  PROC Part13()
    MoveL Offs(pOrigin,150.7,114.4,0.0),vDraw,z1,tPen\WObj:=wPaper;
    MoveL Offs(pOrigin,150.5,114.2,0.0),vDraw,z1,tPen\WObj:=wPaper;
    MoveL Offs(pOrigin,150.5,113.3,0.0),vDraw,z1,tPen\WObj:=wPaper;
    MoveL Offs(pOrigin,150.2,113.0,0.0),vDraw,z1,tPen\WObj:=wPaper;
    MoveL Offs(pOrigin,150.0,113.0,0.0),vDraw,z1,tPen\WObj:=wPaper;
    MoveL Offs(pOrigin,149.8,113.3,0.0),vDraw,z1,tPen\WObj:=wPaper;
    MoveL Offs(pOrigin,149.8,113.7,0.0),vDraw,z1,tPen\WObj:=wPaper;
    MoveL Offs(pOrigin,150.0,114.0,0.0),vDraw,z1,tPen\WObj:=wPaper;
    MoveL Offs(pOrigin,150.0,114.2,0.0),vDraw,z1,tPen\WObj:=wPaper;
    MoveL Offs(pOrigin,149.1,114.2,0.0),vDraw,z1,tPen\WObj:=wPaper;
    MoveL Offs(pOrigin,148.8,114.4,0.0),vDraw,z1,tPen\WObj:=wPaper;
    MoveL Offs(pOrigin,148.1,114.4,0.0),vDraw,z1,tPen\WObj:=wPaper;
    MoveL Offs(pOrigin,147.9,114.7,0.0),vDraw,z1,tPen\WObj:=wPaper;
    MoveL Offs(pOrigin,147.7,114.7,0.0),vDraw,z1,tPen\WObj:=wPaper;
    MoveL Offs(pOrigin,147.4,114.4,0.0),vDraw,z1,tPen\WObj:=wPaper;
    MoveL Offs(pOrigin,147.0,114.4,0.0),vDraw,z1,tPen\WObj:=wPaper;
    MoveL Offs(pOrigin,146.5,114.0,0.0),vDraw,z1,tPen\WObj:=wPaper;
    MoveL Offs(pOrigin,145.8,114.0,0.0),vDraw,z1,tPen\WObj:=wPaper;
    MoveL Offs(pOrigin,145.6,114.2,0.0),vDraw,z1,tPen\WObj:=wPaper;
    MoveL Offs(pOrigin,145.3,114.9,0.0),vDraw,z1,tPen\WObj:=wPaper;
    MoveL Offs(pOrigin,145.1,114.9,0.0),vDraw,z1,tPen\WObj:=wPaper;
    MoveL Offs(pOrigin,144.4,115.4,0.0),vDraw,z1,tPen\WObj:=wPaper;
    MoveL Offs(pOrigin,144.4,115.6,0.0),vDraw,z1,tPen\WObj:=wPaper;
    MoveL Offs(pOrigin,144.2,115.8,0.0),vDraw,z1,tPen\WObj:=wPaper;
    MoveL Offs(pOrigin,144.2,116.5,0.0),vDraw,z1,tPen\WObj:=wPaper;
    MoveL Offs(pOrigin,143.7,117.2,0.0),vDraw,z1,tPen\WObj:=wPaper;
    MoveL Offs(pOrigin,143.7,117.7,0.0),vDraw,z1,tPen\WObj:=wPaper;
    MoveL Offs(pOrigin,143.5,117.9,0.0),vDraw,z1,tPen\WObj:=wPaper;
    MoveL Offs(pOrigin,143.5,118.4,0.0),vDraw,z1,tPen\WObj:=wPaper;
    MoveL Offs(pOrigin,143.2,118.6,0.0),vDraw,z1,tPen\WObj:=wPaper;
    MoveL Offs(pOrigin,143.2,119.6,0.0),vDraw,z1,tPen\WObj:=wPaper;
    MoveL Offs(pOrigin,143.9,120.7,0.0),vDraw,z1,tPen\WObj:=wPaper;
    MoveL Offs(pOrigin,143.9,121.4,0.0),vDraw,z1,tPen\WObj:=wPaper;
    MoveL Offs(pOrigin,144.9,122.1,0.0),vDraw,z1,tPen\WObj:=wPaper;
    MoveL Offs(pOrigin,146.7,120.5,0.0),vDraw,z1,tPen\WObj:=wPaper;
    MoveL Offs(pOrigin,147.9,120.0,0.0),vDraw,z1,tPen\WObj:=wPaper;
    MoveL Offs(pOrigin,148.4,119.6,0.0),vDraw,z1,tPen\WObj:=wPaper;
    MoveL Offs(pOrigin,148.4,119.3,0.0),vDraw,z1,tPen\WObj:=wPaper;
    MoveL Offs(pOrigin,149.3,118.6,0.0),vDraw,fine,tPen\WObj:=wPaper;
    MoveL Offs(pOrigin,149.3,118.6,15.0),vApproach,z5,tPen\WObj:=wPaper;
    MoveL Offs(pOrigin,155.6,113.5,15.0),vTravel,z5,tPen\WObj:=wPaper;
    MoveL Offs(pOrigin,155.6,113.5,0.0),vApproach,fine,tPen\WObj:=wPaper;
    MoveL Offs(pOrigin,156.3,114.2,0.0),vDraw,z1,tPen\WObj:=wPaper;
    MoveL Offs(pOrigin,156.5,114.2,0.0),vDraw,z1,tPen\WObj:=wPaper;
    MoveL Offs(pOrigin,156.8,114.0,0.0),vDraw,z1,tPen\WObj:=wPaper;
    MoveL Offs(pOrigin,156.8,113.5,0.0),vDraw,z1,tPen\WObj:=wPaper;
    MoveL Offs(pOrigin,156.3,112.8,0.0),vDraw,z1,tPen\WObj:=wPaper;
    MoveL Offs(pOrigin,155.8,112.8,0.0),vDraw,z1,tPen\WObj:=wPaper;
    MoveL Offs(pOrigin,155.6,113.0,0.0),vDraw,z1,tPen\WObj:=wPaper;
    MoveL Offs(pOrigin,155.6,113.5,0.0),vDraw,fine,tPen\WObj:=wPaper;
    MoveL Offs(pOrigin,155.6,113.5,15.0),vApproach,z5,tPen\WObj:=wPaper;
    MoveL Offs(pOrigin,163.8,115.6,15.0),vTravel,z5,tPen\WObj:=wPaper;
    MoveL Offs(pOrigin,163.8,115.6,0.0),vApproach,fine,tPen\WObj:=wPaper;
    MoveL Offs(pOrigin,164.0,115.8,0.0),vDraw,z1,tPen\WObj:=wPaper;
    MoveL Offs(pOrigin,164.0,116.1,0.0),vDraw,z1,tPen\WObj:=wPaper;
    MoveL Offs(pOrigin,164.7,116.5,0.0),vDraw,z1,tPen\WObj:=wPaper;
    MoveL Offs(pOrigin,164.7,117.0,0.0),vDraw,z1,tPen\WObj:=wPaper;
    MoveL Offs(pOrigin,164.9,117.2,0.0),vDraw,z1,tPen\WObj:=wPaper;
    MoveL Offs(pOrigin,166.1,117.0,0.0),vDraw,z1,tPen\WObj:=wPaper;
    MoveL Offs(pOrigin,166.6,116.5,0.0),vDraw,z1,tPen\WObj:=wPaper;
    MoveL Offs(pOrigin,166.3,116.3,0.0),vDraw,z1,tPen\WObj:=wPaper;
    MoveL Offs(pOrigin,165.9,116.3,0.0),vDraw,z1,tPen\WObj:=wPaper;
    MoveL Offs(pOrigin,165.9,116.1,0.0),vDraw,z1,tPen\WObj:=wPaper;
    MoveL Offs(pOrigin,165.2,115.4,0.0),vDraw,z1,tPen\WObj:=wPaper;
    MoveL Offs(pOrigin,164.9,115.4,0.0),vDraw,z1,tPen\WObj:=wPaper;
    MoveL Offs(pOrigin,164.7,115.1,0.0),vDraw,z1,tPen\WObj:=wPaper;
    MoveL Offs(pOrigin,164.2,115.1,0.0),vDraw,z1,tPen\WObj:=wPaper;
    MoveL Offs(pOrigin,163.8,115.6,0.0),vDraw,fine,tPen\WObj:=wPaper;
    MoveL Offs(pOrigin,163.8,115.6,15.0),vApproach,z5,tPen\WObj:=wPaper;
    MoveL Offs(pOrigin,180.6,104.4,15.0),vTravel,z5,tPen\WObj:=wPaper;
    MoveL Offs(pOrigin,180.6,104.4,0.0),vApproach,fine,tPen\WObj:=wPaper;
    MoveL Offs(pOrigin,180.6,103.9,0.0),vDraw,z1,tPen\WObj:=wPaper;
    MoveL Offs(pOrigin,180.8,103.7,0.0),vDraw,z1,tPen\WObj:=wPaper;
    MoveL Offs(pOrigin,180.8,102.8,0.0),vDraw,z1,tPen\WObj:=wPaper;
    MoveL Offs(pOrigin,181.0,102.5,0.0),vDraw,z1,tPen\WObj:=wPaper;
    MoveL Offs(pOrigin,181.0,101.6,0.0),vDraw,z1,tPen\WObj:=wPaper;
    MoveL Offs(pOrigin,181.3,101.4,0.0),vDraw,z1,tPen\WObj:=wPaper;
    MoveL Offs(pOrigin,181.3,100.2,0.0),vDraw,z1,tPen\WObj:=wPaper;
    MoveL Offs(pOrigin,181.5,100.0,0.0),vDraw,z1,tPen\WObj:=wPaper;
    MoveL Offs(pOrigin,181.5,97.6,0.0),vDraw,z1,tPen\WObj:=wPaper;
    MoveL Offs(pOrigin,181.7,97.4,0.0),vDraw,z1,tPen\WObj:=wPaper;
    MoveL Offs(pOrigin,181.7,96.7,0.0),vDraw,z1,tPen\WObj:=wPaper;
    MoveL Offs(pOrigin,181.5,96.5,0.0),vDraw,z1,tPen\WObj:=wPaper;
    MoveL Offs(pOrigin,181.5,92.3,0.0),vDraw,z1,tPen\WObj:=wPaper;
    MoveL Offs(pOrigin,181.3,92.0,0.0),vDraw,z1,tPen\WObj:=wPaper;
    MoveL Offs(pOrigin,181.3,90.6,0.0),vDraw,z1,tPen\WObj:=wPaper;
    MoveL Offs(pOrigin,181.0,90.4,0.0),vDraw,z1,tPen\WObj:=wPaper;
    MoveL Offs(pOrigin,181.0,89.7,0.0),vDraw,z1,tPen\WObj:=wPaper;
    MoveL Offs(pOrigin,180.8,89.5,0.0),vDraw,z1,tPen\WObj:=wPaper;
    MoveL Offs(pOrigin,180.8,89.0,0.0),vDraw,z1,tPen\WObj:=wPaper;
    MoveL Offs(pOrigin,180.6,88.8,0.0),vDraw,z1,tPen\WObj:=wPaper;
    MoveL Offs(pOrigin,180.6,88.1,0.0),vDraw,z1,tPen\WObj:=wPaper;
    MoveL Offs(pOrigin,180.3,87.8,0.0),vDraw,z1,tPen\WObj:=wPaper;
    MoveL Offs(pOrigin,180.3,86.9,0.0),vDraw,z1,tPen\WObj:=wPaper;
    MoveL Offs(pOrigin,180.1,86.7,0.0),vDraw,z1,tPen\WObj:=wPaper;
    MoveL Offs(pOrigin,180.1,86.0,0.0),vDraw,z1,tPen\WObj:=wPaper;
    MoveL Offs(pOrigin,179.9,85.7,0.0),vDraw,z1,tPen\WObj:=wPaper;
    MoveL Offs(pOrigin,179.9,85.0,0.0),vDraw,z1,tPen\WObj:=wPaper;
    MoveL Offs(pOrigin,179.6,84.8,0.0),vDraw,z1,tPen\WObj:=wPaper;
    MoveL Offs(pOrigin,179.6,83.9,0.0),vDraw,z1,tPen\WObj:=wPaper;
    MoveL Offs(pOrigin,179.4,83.6,0.0),vDraw,z1,tPen\WObj:=wPaper;
    MoveL Offs(pOrigin,179.4,82.5,0.0),vDraw,z1,tPen\WObj:=wPaper;
    MoveL Offs(pOrigin,179.2,82.2,0.0),vDraw,z1,tPen\WObj:=wPaper;
    MoveL Offs(pOrigin,179.2,81.1,0.0),vDraw,z1,tPen\WObj:=wPaper;
    MoveL Offs(pOrigin,178.9,80.8,0.0),vDraw,z1,tPen\WObj:=wPaper;
    MoveL Offs(pOrigin,178.9,79.7,0.0),vDraw,z1,tPen\WObj:=wPaper;
    MoveL Offs(pOrigin,178.7,79.4,0.0),vDraw,z1,tPen\WObj:=wPaper;
    MoveL Offs(pOrigin,178.7,78.0,0.0),vDraw,z1,tPen\WObj:=wPaper;
    MoveL Offs(pOrigin,178.5,77.8,0.0),vDraw,z1,tPen\WObj:=wPaper;
    MoveL Offs(pOrigin,178.5,76.4,0.0),vDraw,z1,tPen\WObj:=wPaper;
    MoveL Offs(pOrigin,178.2,76.2,0.0),vDraw,z1,tPen\WObj:=wPaper;
    MoveL Offs(pOrigin,178.2,75.5,0.0),vDraw,z1,tPen\WObj:=wPaper;
    MoveL Offs(pOrigin,178.0,75.2,0.0),vDraw,z1,tPen\WObj:=wPaper;
    MoveL Offs(pOrigin,178.0,74.3,0.0),vDraw,z1,tPen\WObj:=wPaper;
    MoveL Offs(pOrigin,177.8,74.1,0.0),vDraw,z1,tPen\WObj:=wPaper;
    MoveL Offs(pOrigin,177.8,72.4,0.0),vDraw,z1,tPen\WObj:=wPaper;
    MoveL Offs(pOrigin,177.5,72.2,0.0),vDraw,z1,tPen\WObj:=wPaper;
    MoveL Offs(pOrigin,177.5,71.7,0.0),vDraw,z1,tPen\WObj:=wPaper;
    MoveL Offs(pOrigin,177.3,71.5,0.0),vDraw,z1,tPen\WObj:=wPaper;
    MoveL Offs(pOrigin,177.3,70.3,0.0),vDraw,z1,tPen\WObj:=wPaper;
  ENDPROC

  PROC Part14()
    MoveL Offs(pOrigin,177.1,70.1,0.0),vDraw,z1,tPen\WObj:=wPaper;
    MoveL Offs(pOrigin,177.1,69.2,0.0),vDraw,z1,tPen\WObj:=wPaper;
    MoveL Offs(pOrigin,176.8,68.9,0.0),vDraw,z1,tPen\WObj:=wPaper;
    MoveL Offs(pOrigin,176.8,67.8,0.0),vDraw,z1,tPen\WObj:=wPaper;
    MoveL Offs(pOrigin,176.6,67.5,0.0),vDraw,z1,tPen\WObj:=wPaper;
    MoveL Offs(pOrigin,176.6,66.4,0.0),vDraw,z1,tPen\WObj:=wPaper;
    MoveL Offs(pOrigin,176.4,66.1,0.0),vDraw,z1,tPen\WObj:=wPaper;
    MoveL Offs(pOrigin,176.4,65.2,0.0),vDraw,z1,tPen\WObj:=wPaper;
    MoveL Offs(pOrigin,176.1,65.0,0.0),vDraw,z1,tPen\WObj:=wPaper;
    MoveL Offs(pOrigin,176.1,64.0,0.0),vDraw,z1,tPen\WObj:=wPaper;
    MoveL Offs(pOrigin,175.9,63.8,0.0),vDraw,z1,tPen\WObj:=wPaper;
    MoveL Offs(pOrigin,175.9,62.6,0.0),vDraw,z1,tPen\WObj:=wPaper;
    MoveL Offs(pOrigin,175.7,62.4,0.0),vDraw,z1,tPen\WObj:=wPaper;
    MoveL Offs(pOrigin,175.7,61.5,0.0),vDraw,z1,tPen\WObj:=wPaper;
    MoveL Offs(pOrigin,175.4,61.2,0.0),vDraw,z1,tPen\WObj:=wPaper;
    MoveL Offs(pOrigin,175.4,60.5,0.0),vDraw,z1,tPen\WObj:=wPaper;
    MoveL Offs(pOrigin,175.2,60.3,0.0),vDraw,z1,tPen\WObj:=wPaper;
    MoveL Offs(pOrigin,175.2,59.1,0.0),vDraw,z1,tPen\WObj:=wPaper;
    MoveL Offs(pOrigin,175.0,58.9,0.0),vDraw,z1,tPen\WObj:=wPaper;
    MoveL Offs(pOrigin,175.0,58.0,0.0),vDraw,z1,tPen\WObj:=wPaper;
    MoveL Offs(pOrigin,174.7,57.7,0.0),vDraw,z1,tPen\WObj:=wPaper;
    MoveL Offs(pOrigin,174.7,57.0,0.0),vDraw,z1,tPen\WObj:=wPaper;
    MoveL Offs(pOrigin,174.5,56.8,0.0),vDraw,z1,tPen\WObj:=wPaper;
    MoveL Offs(pOrigin,174.5,55.9,0.0),vDraw,z1,tPen\WObj:=wPaper;
    MoveL Offs(pOrigin,174.3,55.6,0.0),vDraw,z1,tPen\WObj:=wPaper;
    MoveL Offs(pOrigin,174.3,54.7,0.0),vDraw,z1,tPen\WObj:=wPaper;
    MoveL Offs(pOrigin,174.0,54.5,0.0),vDraw,z1,tPen\WObj:=wPaper;
    MoveL Offs(pOrigin,174.0,53.8,0.0),vDraw,z1,tPen\WObj:=wPaper;
    MoveL Offs(pOrigin,173.8,53.5,0.0),vDraw,z1,tPen\WObj:=wPaper;
    MoveL Offs(pOrigin,173.8,52.6,0.0),vDraw,z1,tPen\WObj:=wPaper;
    MoveL Offs(pOrigin,173.6,52.4,0.0),vDraw,z1,tPen\WObj:=wPaper;
    MoveL Offs(pOrigin,173.6,51.7,0.0),vDraw,z1,tPen\WObj:=wPaper;
    MoveL Offs(pOrigin,173.3,51.4,0.0),vDraw,z1,tPen\WObj:=wPaper;
    MoveL Offs(pOrigin,173.3,50.5,0.0),vDraw,z1,tPen\WObj:=wPaper;
    MoveL Offs(pOrigin,173.1,50.3,0.0),vDraw,z1,tPen\WObj:=wPaper;
    MoveL Offs(pOrigin,173.1,49.6,0.0),vDraw,z1,tPen\WObj:=wPaper;
    MoveL Offs(pOrigin,172.9,49.3,0.0),vDraw,z1,tPen\WObj:=wPaper;
    MoveL Offs(pOrigin,172.9,48.4,0.0),vDraw,z1,tPen\WObj:=wPaper;
    MoveL Offs(pOrigin,172.6,48.2,0.0),vDraw,z1,tPen\WObj:=wPaper;
    MoveL Offs(pOrigin,172.6,47.2,0.0),vDraw,z1,tPen\WObj:=wPaper;
    MoveL Offs(pOrigin,172.4,47.0,0.0),vDraw,z1,tPen\WObj:=wPaper;
    MoveL Offs(pOrigin,172.4,46.1,0.0),vDraw,z1,tPen\WObj:=wPaper;
    MoveL Offs(pOrigin,172.2,45.8,0.0),vDraw,z1,tPen\WObj:=wPaper;
    MoveL Offs(pOrigin,172.2,44.9,0.0),vDraw,z1,tPen\WObj:=wPaper;
    MoveL Offs(pOrigin,171.9,44.7,0.0),vDraw,z1,tPen\WObj:=wPaper;
    MoveL Offs(pOrigin,171.9,44.0,0.0),vDraw,z1,tPen\WObj:=wPaper;
    MoveL Offs(pOrigin,171.7,43.7,0.0),vDraw,z1,tPen\WObj:=wPaper;
    MoveL Offs(pOrigin,171.7,43.0,0.0),vDraw,z1,tPen\WObj:=wPaper;
    MoveL Offs(pOrigin,171.5,42.8,0.0),vDraw,z1,tPen\WObj:=wPaper;
    MoveL Offs(pOrigin,171.5,41.9,0.0),vDraw,z1,tPen\WObj:=wPaper;
    MoveL Offs(pOrigin,171.2,41.6,0.0),vDraw,z1,tPen\WObj:=wPaper;
    MoveL Offs(pOrigin,171.2,40.9,0.0),vDraw,z1,tPen\WObj:=wPaper;
    MoveL Offs(pOrigin,171.0,40.7,0.0),vDraw,z1,tPen\WObj:=wPaper;
    MoveL Offs(pOrigin,171.0,39.8,0.0),vDraw,z1,tPen\WObj:=wPaper;
    MoveL Offs(pOrigin,170.8,39.5,0.0),vDraw,z1,tPen\WObj:=wPaper;
    MoveL Offs(pOrigin,170.8,38.8,0.0),vDraw,z1,tPen\WObj:=wPaper;
    MoveL Offs(pOrigin,170.5,38.6,0.0),vDraw,z1,tPen\WObj:=wPaper;
    MoveL Offs(pOrigin,170.5,37.7,0.0),vDraw,z1,tPen\WObj:=wPaper;
    MoveL Offs(pOrigin,170.3,37.4,0.0),vDraw,z1,tPen\WObj:=wPaper;
    MoveL Offs(pOrigin,170.3,36.7,0.0),vDraw,z1,tPen\WObj:=wPaper;
    MoveL Offs(pOrigin,170.1,36.5,0.0),vDraw,z1,tPen\WObj:=wPaper;
    MoveL Offs(pOrigin,170.1,35.8,0.0),vDraw,z1,tPen\WObj:=wPaper;
    MoveL Offs(pOrigin,169.8,35.6,0.0),vDraw,z1,tPen\WObj:=wPaper;
    MoveL Offs(pOrigin,169.8,34.9,0.0),vDraw,z1,tPen\WObj:=wPaper;
    MoveL Offs(pOrigin,169.6,34.6,0.0),vDraw,z1,tPen\WObj:=wPaper;
    MoveL Offs(pOrigin,169.6,33.7,0.0),vDraw,z1,tPen\WObj:=wPaper;
    MoveL Offs(pOrigin,169.4,33.5,0.0),vDraw,z1,tPen\WObj:=wPaper;
    MoveL Offs(pOrigin,169.4,32.8,0.0),vDraw,z1,tPen\WObj:=wPaper;
    MoveL Offs(pOrigin,169.1,32.5,0.0),vDraw,z1,tPen\WObj:=wPaper;
    MoveL Offs(pOrigin,169.1,31.8,0.0),vDraw,z1,tPen\WObj:=wPaper;
    MoveL Offs(pOrigin,168.9,31.6,0.0),vDraw,z1,tPen\WObj:=wPaper;
    MoveL Offs(pOrigin,168.9,30.9,0.0),vDraw,z1,tPen\WObj:=wPaper;
    MoveL Offs(pOrigin,168.7,30.7,0.0),vDraw,z1,tPen\WObj:=wPaper;
    MoveL Offs(pOrigin,168.7,29.7,0.0),vDraw,z1,tPen\WObj:=wPaper;
    MoveL Offs(pOrigin,168.4,29.5,0.0),vDraw,z1,tPen\WObj:=wPaper;
    MoveL Offs(pOrigin,168.4,28.8,0.0),vDraw,z1,tPen\WObj:=wPaper;
    MoveL Offs(pOrigin,168.2,28.6,0.0),vDraw,z1,tPen\WObj:=wPaper;
    MoveL Offs(pOrigin,168.2,27.6,0.0),vDraw,z1,tPen\WObj:=wPaper;
    MoveL Offs(pOrigin,168.0,27.4,0.0),vDraw,z1,tPen\WObj:=wPaper;
    MoveL Offs(pOrigin,168.0,26.9,0.0),vDraw,z1,tPen\WObj:=wPaper;
    MoveL Offs(pOrigin,167.7,26.7,0.0),vDraw,z1,tPen\WObj:=wPaper;
    MoveL Offs(pOrigin,167.7,25.8,0.0),vDraw,z1,tPen\WObj:=wPaper;
    MoveL Offs(pOrigin,167.5,25.5,0.0),vDraw,z1,tPen\WObj:=wPaper;
    MoveL Offs(pOrigin,167.5,24.8,0.0),vDraw,z1,tPen\WObj:=wPaper;
    MoveL Offs(pOrigin,167.3,24.6,0.0),vDraw,z1,tPen\WObj:=wPaper;
    MoveL Offs(pOrigin,167.3,23.9,0.0),vDraw,z1,tPen\WObj:=wPaper;
    MoveL Offs(pOrigin,167.0,23.7,0.0),vDraw,z1,tPen\WObj:=wPaper;
    MoveL Offs(pOrigin,167.0,23.0,0.0),vDraw,z1,tPen\WObj:=wPaper;
    MoveL Offs(pOrigin,166.8,22.7,0.0),vDraw,z1,tPen\WObj:=wPaper;
    MoveL Offs(pOrigin,166.8,22.0,0.0),vDraw,z1,tPen\WObj:=wPaper;
    MoveL Offs(pOrigin,166.6,21.8,0.0),vDraw,z1,tPen\WObj:=wPaper;
    MoveL Offs(pOrigin,166.6,21.1,0.0),vDraw,z1,tPen\WObj:=wPaper;
    MoveL Offs(pOrigin,166.3,20.9,0.0),vDraw,z1,tPen\WObj:=wPaper;
    MoveL Offs(pOrigin,166.3,20.2,0.0),vDraw,z1,tPen\WObj:=wPaper;
    MoveL Offs(pOrigin,166.1,19.9,0.0),vDraw,z1,tPen\WObj:=wPaper;
    MoveL Offs(pOrigin,166.1,19.5,0.0),vDraw,z1,tPen\WObj:=wPaper;
    MoveL Offs(pOrigin,165.9,19.2,0.0),vDraw,z1,tPen\WObj:=wPaper;
    MoveL Offs(pOrigin,165.9,18.3,0.0),vDraw,z1,tPen\WObj:=wPaper;
    MoveL Offs(pOrigin,165.6,18.1,0.0),vDraw,z1,tPen\WObj:=wPaper;
    MoveL Offs(pOrigin,165.6,17.6,0.0),vDraw,z1,tPen\WObj:=wPaper;
    MoveL Offs(pOrigin,165.4,17.4,0.0),vDraw,z1,tPen\WObj:=wPaper;
    MoveL Offs(pOrigin,165.4,16.7,0.0),vDraw,z1,tPen\WObj:=wPaper;
    MoveL Offs(pOrigin,165.2,16.4,0.0),vDraw,z1,tPen\WObj:=wPaper;
    MoveL Offs(pOrigin,165.2,15.7,0.0),vDraw,z1,tPen\WObj:=wPaper;
    MoveL Offs(pOrigin,164.9,15.5,0.0),vDraw,z1,tPen\WObj:=wPaper;
    MoveL Offs(pOrigin,164.9,14.8,0.0),vDraw,z1,tPen\WObj:=wPaper;
    MoveL Offs(pOrigin,164.7,14.6,0.0),vDraw,z1,tPen\WObj:=wPaper;
    MoveL Offs(pOrigin,164.7,13.9,0.0),vDraw,z1,tPen\WObj:=wPaper;
    MoveL Offs(pOrigin,164.5,13.6,0.0),vDraw,z1,tPen\WObj:=wPaper;
    MoveL Offs(pOrigin,164.5,12.9,0.0),vDraw,z1,tPen\WObj:=wPaper;
    MoveL Offs(pOrigin,164.2,12.7,0.0),vDraw,z1,tPen\WObj:=wPaper;
    MoveL Offs(pOrigin,164.2,12.0,0.0),vDraw,z1,tPen\WObj:=wPaper;
    MoveL Offs(pOrigin,164.0,11.8,0.0),vDraw,z1,tPen\WObj:=wPaper;
    MoveL Offs(pOrigin,164.0,11.1,0.0),vDraw,z1,tPen\WObj:=wPaper;
    MoveL Offs(pOrigin,163.8,10.8,0.0),vDraw,z1,tPen\WObj:=wPaper;
    MoveL Offs(pOrigin,163.8,10.1,0.0),vDraw,z1,tPen\WObj:=wPaper;
    MoveL Offs(pOrigin,163.5,9.9,0.0),vDraw,z1,tPen\WObj:=wPaper;
    MoveL Offs(pOrigin,163.5,9.4,0.0),vDraw,z1,tPen\WObj:=wPaper;
    MoveL Offs(pOrigin,163.3,9.2,0.0),vDraw,z1,tPen\WObj:=wPaper;
    MoveL Offs(pOrigin,163.3,8.5,0.0),vDraw,z1,tPen\WObj:=wPaper;
  ENDPROC

  PROC Part15()
    MoveL Offs(pOrigin,163.1,8.3,0.0),vDraw,z1,tPen\WObj:=wPaper;
    MoveL Offs(pOrigin,163.1,7.6,0.0),vDraw,z1,tPen\WObj:=wPaper;
    MoveL Offs(pOrigin,162.8,7.3,0.0),vDraw,z1,tPen\WObj:=wPaper;
    MoveL Offs(pOrigin,162.8,6.6,0.0),vDraw,z1,tPen\WObj:=wPaper;
    MoveL Offs(pOrigin,162.6,6.4,0.0),vDraw,z1,tPen\WObj:=wPaper;
    MoveL Offs(pOrigin,162.6,5.7,0.0),vDraw,z1,tPen\WObj:=wPaper;
    MoveL Offs(pOrigin,162.4,5.5,0.0),vDraw,z1,tPen\WObj:=wPaper;
    MoveL Offs(pOrigin,162.4,5.2,0.0),vDraw,z1,tPen\WObj:=wPaper;
    MoveL Offs(pOrigin,231.7,5.2,0.0),vDraw,z1,tPen\WObj:=wPaper;
    MoveL Offs(pOrigin,231.7,78.5,0.0),vDraw,z1,tPen\WObj:=wPaper;
    MoveL Offs(pOrigin,230.7,78.5,0.0),vDraw,z1,tPen\WObj:=wPaper;
    MoveL Offs(pOrigin,230.5,78.3,0.0),vDraw,z1,tPen\WObj:=wPaper;
    MoveL Offs(pOrigin,230.0,78.3,0.0),vDraw,z1,tPen\WObj:=wPaper;
    MoveL Offs(pOrigin,229.3,79.0,0.0),vDraw,z1,tPen\WObj:=wPaper;
    MoveL Offs(pOrigin,229.1,79.0,0.0),vDraw,z1,tPen\WObj:=wPaper;
    MoveL Offs(pOrigin,227.0,80.1,0.0),vDraw,z1,tPen\WObj:=wPaper;
    MoveL Offs(pOrigin,226.5,80.1,0.0),vDraw,z1,tPen\WObj:=wPaper;
    MoveL Offs(pOrigin,225.4,80.8,0.0),vDraw,z1,tPen\WObj:=wPaper;
    MoveL Offs(pOrigin,224.9,80.8,0.0),vDraw,z1,tPen\WObj:=wPaper;
    MoveL Offs(pOrigin,224.2,81.3,0.0),vDraw,z1,tPen\WObj:=wPaper;
    MoveL Offs(pOrigin,223.7,81.3,0.0),vDraw,z1,tPen\WObj:=wPaper;
    MoveL Offs(pOrigin,223.0,81.8,0.0),vDraw,z1,tPen\WObj:=wPaper;
    MoveL Offs(pOrigin,222.6,81.8,0.0),vDraw,z1,tPen\WObj:=wPaper;
    MoveL Offs(pOrigin,222.3,82.0,0.0),vDraw,z1,tPen\WObj:=wPaper;
    MoveL Offs(pOrigin,222.1,82.0,0.0),vDraw,z1,tPen\WObj:=wPaper;
    MoveL Offs(pOrigin,221.4,82.5,0.0),vDraw,z1,tPen\WObj:=wPaper;
    MoveL Offs(pOrigin,220.9,82.5,0.0),vDraw,z1,tPen\WObj:=wPaper;
    MoveL Offs(pOrigin,220.2,82.9,0.0),vDraw,z1,tPen\WObj:=wPaper;
    MoveL Offs(pOrigin,219.1,83.2,0.0),vDraw,z1,tPen\WObj:=wPaper;
    MoveL Offs(pOrigin,218.4,83.6,0.0),vDraw,z1,tPen\WObj:=wPaper;
    MoveL Offs(pOrigin,217.2,83.9,0.0),vDraw,z1,tPen\WObj:=wPaper;
    MoveL Offs(pOrigin,216.5,84.3,0.0),vDraw,z1,tPen\WObj:=wPaper;
    MoveL Offs(pOrigin,216.0,84.3,0.0),vDraw,z1,tPen\WObj:=wPaper;
    MoveL Offs(pOrigin,215.3,84.8,0.0),vDraw,z1,tPen\WObj:=wPaper;
    MoveL Offs(pOrigin,214.9,84.8,0.0),vDraw,z1,tPen\WObj:=wPaper;
    MoveL Offs(pOrigin,214.6,85.0,0.0),vDraw,z1,tPen\WObj:=wPaper;
    MoveL Offs(pOrigin,213.5,85.3,0.0),vDraw,z1,tPen\WObj:=wPaper;
    MoveL Offs(pOrigin,212.8,85.7,0.0),vDraw,z1,tPen\WObj:=wPaper;
    MoveL Offs(pOrigin,212.3,85.7,0.0),vDraw,z1,tPen\WObj:=wPaper;
    MoveL Offs(pOrigin,212.1,86.0,0.0),vDraw,z1,tPen\WObj:=wPaper;
    MoveL Offs(pOrigin,210.9,86.2,0.0),vDraw,z1,tPen\WObj:=wPaper;
    MoveL Offs(pOrigin,210.2,86.7,0.0),vDraw,z1,tPen\WObj:=wPaper;
    MoveL Offs(pOrigin,209.7,86.7,0.0),vDraw,z1,tPen\WObj:=wPaper;
    MoveL Offs(pOrigin,209.5,86.9,0.0),vDraw,z1,tPen\WObj:=wPaper;
    MoveL Offs(pOrigin,208.3,87.1,0.0),vDraw,z1,tPen\WObj:=wPaper;
    MoveL Offs(pOrigin,207.6,87.6,0.0),vDraw,z1,tPen\WObj:=wPaper;
    MoveL Offs(pOrigin,207.2,87.6,0.0),vDraw,z1,tPen\WObj:=wPaper;
    MoveL Offs(pOrigin,206.9,87.8,0.0),vDraw,z1,tPen\WObj:=wPaper;
    MoveL Offs(pOrigin,205.8,88.1,0.0),vDraw,z1,tPen\WObj:=wPaper;
    MoveL Offs(pOrigin,205.5,88.3,0.0),vDraw,z1,tPen\WObj:=wPaper;
    MoveL Offs(pOrigin,205.3,88.3,0.0),vDraw,z1,tPen\WObj:=wPaper;
    MoveL Offs(pOrigin,205.1,88.5,0.0),vDraw,z1,tPen\WObj:=wPaper;
    MoveL Offs(pOrigin,204.6,88.5,0.0),vDraw,z1,tPen\WObj:=wPaper;
    MoveL Offs(pOrigin,203.9,89.0,0.0),vDraw,z1,tPen\WObj:=wPaper;
    MoveL Offs(pOrigin,203.4,89.0,0.0),vDraw,z1,tPen\WObj:=wPaper;
    MoveL Offs(pOrigin,203.2,89.2,0.0),vDraw,z1,tPen\WObj:=wPaper;
    MoveL Offs(pOrigin,202.7,89.2,0.0),vDraw,z1,tPen\WObj:=wPaper;
    MoveL Offs(pOrigin,202.0,89.7,0.0),vDraw,z1,tPen\WObj:=wPaper;
    MoveL Offs(pOrigin,200.9,89.9,0.0),vDraw,z1,tPen\WObj:=wPaper;
    MoveL Offs(pOrigin,200.2,90.4,0.0),vDraw,z1,tPen\WObj:=wPaper;
    MoveL Offs(pOrigin,199.7,90.4,0.0),vDraw,z1,tPen\WObj:=wPaper;
    MoveL Offs(pOrigin,199.0,90.9,0.0),vDraw,z1,tPen\WObj:=wPaper;
    MoveL Offs(pOrigin,198.5,90.9,0.0),vDraw,z1,tPen\WObj:=wPaper;
    MoveL Offs(pOrigin,198.3,91.1,0.0),vDraw,z1,tPen\WObj:=wPaper;
    MoveL Offs(pOrigin,197.8,91.1,0.0),vDraw,z1,tPen\WObj:=wPaper;
    MoveL Offs(pOrigin,197.1,91.6,0.0),vDraw,z1,tPen\WObj:=wPaper;
    MoveL Offs(pOrigin,196.0,91.8,0.0),vDraw,z1,tPen\WObj:=wPaper;
    MoveL Offs(pOrigin,195.3,92.3,0.0),vDraw,z1,tPen\WObj:=wPaper;
    MoveL Offs(pOrigin,194.1,92.5,0.0),vDraw,z1,tPen\WObj:=wPaper;
    MoveL Offs(pOrigin,193.4,93.0,0.0),vDraw,z1,tPen\WObj:=wPaper;
    MoveL Offs(pOrigin,192.9,93.0,0.0),vDraw,z1,tPen\WObj:=wPaper;
    MoveL Offs(pOrigin,192.7,93.2,0.0),vDraw,z1,tPen\WObj:=wPaper;
    MoveL Offs(pOrigin,191.5,93.4,0.0),vDraw,z1,tPen\WObj:=wPaper;
    MoveL Offs(pOrigin,191.1,93.9,0.0),vDraw,z1,tPen\WObj:=wPaper;
    MoveL Offs(pOrigin,190.8,93.9,0.0),vDraw,z1,tPen\WObj:=wPaper;
    MoveL Offs(pOrigin,189.9,94.8,0.0),vDraw,z1,tPen\WObj:=wPaper;
    MoveL Offs(pOrigin,189.7,94.8,0.0),vDraw,z1,tPen\WObj:=wPaper;
    MoveL Offs(pOrigin,189.0,95.5,0.0),vDraw,z1,tPen\WObj:=wPaper;
    MoveL Offs(pOrigin,188.7,95.5,0.0),vDraw,z1,tPen\WObj:=wPaper;
    MoveL Offs(pOrigin,187.3,96.9,0.0),vDraw,z1,tPen\WObj:=wPaper;
    MoveL Offs(pOrigin,187.1,96.9,0.0),vDraw,z1,tPen\WObj:=wPaper;
    MoveL Offs(pOrigin,184.1,100.0,0.0),vDraw,z1,tPen\WObj:=wPaper;
    MoveL Offs(pOrigin,184.1,100.2,0.0),vDraw,z1,tPen\WObj:=wPaper;
    MoveL Offs(pOrigin,182.9,101.6,0.0),vDraw,z1,tPen\WObj:=wPaper;
    MoveL Offs(pOrigin,182.7,102.3,0.0),vDraw,z1,tPen\WObj:=wPaper;
    MoveL Offs(pOrigin,182.0,103.0,0.0),vDraw,z1,tPen\WObj:=wPaper;
    MoveL Offs(pOrigin,182.0,103.2,0.0),vDraw,z1,tPen\WObj:=wPaper;
    MoveL Offs(pOrigin,181.3,103.9,0.0),vDraw,z1,tPen\WObj:=wPaper;
    MoveL Offs(pOrigin,181.3,104.2,0.0),vDraw,z1,tPen\WObj:=wPaper;
    MoveL Offs(pOrigin,181.0,104.4,0.0),vDraw,z1,tPen\WObj:=wPaper;
    MoveL Offs(pOrigin,180.6,104.4,0.0),vDraw,fine,tPen\WObj:=wPaper;
    MoveL Offs(pOrigin,180.6,104.4,15.0),vApproach,z5,tPen\WObj:=wPaper;
    MoveL Offs(pOrigin,154.9,77.3,15.0),vTravel,z5,tPen\WObj:=wPaper;
    MoveL Offs(pOrigin,154.9,77.3,0.0),vApproach,fine,tPen\WObj:=wPaper;
    MoveL Offs(pOrigin,155.4,76.9,0.0),vDraw,z1,tPen\WObj:=wPaper;
    MoveL Offs(pOrigin,155.4,76.4,0.0),vDraw,z1,tPen\WObj:=wPaper;
    MoveL Offs(pOrigin,155.1,76.2,0.0),vDraw,z1,tPen\WObj:=wPaper;
    MoveL Offs(pOrigin,154.7,76.2,0.0),vDraw,z1,tPen\WObj:=wPaper;
    MoveL Offs(pOrigin,154.4,76.4,0.0),vDraw,z1,tPen\WObj:=wPaper;
    MoveL Offs(pOrigin,154.4,77.1,0.0),vDraw,z1,tPen\WObj:=wPaper;
    MoveL Offs(pOrigin,154.7,77.3,0.0),vDraw,z1,tPen\WObj:=wPaper;
    MoveL Offs(pOrigin,154.9,77.3,0.0),vDraw,fine,tPen\WObj:=wPaper;
    MoveL Offs(pOrigin,154.9,77.3,15.0),vApproach,z5,tPen\WObj:=wPaper;
    MoveL Offs(pOrigin,153.0,76.4,15.0),vTravel,z5,tPen\WObj:=wPaper;
    MoveL Offs(pOrigin,153.0,76.4,0.0),vApproach,fine,tPen\WObj:=wPaper;
    MoveL Offs(pOrigin,153.0,76.2,0.0),vDraw,z1,tPen\WObj:=wPaper;
    MoveL Offs(pOrigin,152.8,75.9,0.0),vDraw,z1,tPen\WObj:=wPaper;
    MoveL Offs(pOrigin,152.1,76.2,0.0),vDraw,z1,tPen\WObj:=wPaper;
    MoveL Offs(pOrigin,151.4,76.9,0.0),vDraw,z1,tPen\WObj:=wPaper;
    MoveL Offs(pOrigin,151.4,77.1,0.0),vDraw,z1,tPen\WObj:=wPaper;
    MoveL Offs(pOrigin,151.9,77.6,0.0),vDraw,z1,tPen\WObj:=wPaper;
    MoveL Offs(pOrigin,152.1,77.6,0.0),vDraw,z1,tPen\WObj:=wPaper;
    MoveL Offs(pOrigin,152.6,77.1,0.0),vDraw,z1,tPen\WObj:=wPaper;
    MoveL Offs(pOrigin,152.6,76.9,0.0),vDraw,z1,tPen\WObj:=wPaper;
    MoveL Offs(pOrigin,153.0,76.4,0.0),vDraw,fine,tPen\WObj:=wPaper;
    MoveL Offs(pOrigin,153.0,76.4,15.0),vApproach,z5,tPen\WObj:=wPaper;
    MoveL Offs(pOrigin,148.4,82.9,15.0),vTravel,z5,tPen\WObj:=wPaper;
    MoveL Offs(pOrigin,148.4,82.9,0.0),vApproach,fine,tPen\WObj:=wPaper;
    MoveL Offs(pOrigin,147.4,82.9,0.0),vDraw,z1,tPen\WObj:=wPaper;
    MoveL Offs(pOrigin,147.0,83.4,0.0),vDraw,z1,tPen\WObj:=wPaper;
  ENDPROC

  PROC Part16()
    MoveL Offs(pOrigin,147.0,83.9,0.0),vDraw,z1,tPen\WObj:=wPaper;
    MoveL Offs(pOrigin,147.2,84.1,0.0),vDraw,z1,tPen\WObj:=wPaper;
    MoveL Offs(pOrigin,147.2,84.3,0.0),vDraw,z1,tPen\WObj:=wPaper;
    MoveL Offs(pOrigin,147.0,84.6,0.0),vDraw,z1,tPen\WObj:=wPaper;
    MoveL Offs(pOrigin,147.0,85.0,0.0),vDraw,z1,tPen\WObj:=wPaper;
    MoveL Offs(pOrigin,146.7,85.3,0.0),vDraw,z1,tPen\WObj:=wPaper;
    MoveL Offs(pOrigin,146.0,85.3,0.0),vDraw,z1,tPen\WObj:=wPaper;
    MoveL Offs(pOrigin,145.6,84.8,0.0),vDraw,z1,tPen\WObj:=wPaper;
    MoveL Offs(pOrigin,144.9,84.8,0.0),vDraw,z1,tPen\WObj:=wPaper;
    MoveL Offs(pOrigin,144.6,85.0,0.0),vDraw,z1,tPen\WObj:=wPaper;
    MoveL Offs(pOrigin,144.4,85.0,0.0),vDraw,z1,tPen\WObj:=wPaper;
    MoveL Offs(pOrigin,143.2,86.2,0.0),vDraw,z1,tPen\WObj:=wPaper;
    MoveL Offs(pOrigin,143.0,86.2,0.0),vDraw,z1,tPen\WObj:=wPaper;
    MoveL Offs(pOrigin,142.5,86.7,0.0),vDraw,z1,tPen\WObj:=wPaper;
    MoveL Offs(pOrigin,142.1,86.7,0.0),vDraw,z1,tPen\WObj:=wPaper;
    MoveL Offs(pOrigin,140.0,89.0,0.0),vDraw,z1,tPen\WObj:=wPaper;
    MoveL Offs(pOrigin,140.0,89.2,0.0),vDraw,z1,tPen\WObj:=wPaper;
    MoveL Offs(pOrigin,139.7,89.5,0.0),vDraw,z1,tPen\WObj:=wPaper;
    MoveL Offs(pOrigin,139.7,89.9,0.0),vDraw,z1,tPen\WObj:=wPaper;
    MoveL Offs(pOrigin,140.0,90.2,0.0),vDraw,z1,tPen\WObj:=wPaper;
    MoveL Offs(pOrigin,140.2,90.2,0.0),vDraw,z1,tPen\WObj:=wPaper;
    MoveL Offs(pOrigin,140.4,89.9,0.0),vDraw,z1,tPen\WObj:=wPaper;
    MoveL Offs(pOrigin,141.1,89.9,0.0),vDraw,z1,tPen\WObj:=wPaper;
    MoveL Offs(pOrigin,141.6,89.5,0.0),vDraw,z1,tPen\WObj:=wPaper;
    MoveL Offs(pOrigin,142.3,89.2,0.0),vDraw,z1,tPen\WObj:=wPaper;
    MoveL Offs(pOrigin,143.5,88.1,0.0),vDraw,z1,tPen\WObj:=wPaper;
    MoveL Offs(pOrigin,144.2,87.8,0.0),vDraw,z1,tPen\WObj:=wPaper;
    MoveL Offs(pOrigin,144.9,87.1,0.0),vDraw,z1,tPen\WObj:=wPaper;
    MoveL Offs(pOrigin,145.6,87.1,0.0),vDraw,z1,tPen\WObj:=wPaper;
    MoveL Offs(pOrigin,146.0,86.7,0.0),vDraw,z1,tPen\WObj:=wPaper;
    MoveL Offs(pOrigin,146.7,86.4,0.0),vDraw,z1,tPen\WObj:=wPaper;
    MoveL Offs(pOrigin,147.9,85.3,0.0),vDraw,z1,tPen\WObj:=wPaper;
    MoveL Offs(pOrigin,148.1,85.3,0.0),vDraw,z1,tPen\WObj:=wPaper;
    MoveL Offs(pOrigin,148.6,84.8,0.0),vDraw,z1,tPen\WObj:=wPaper;
    MoveL Offs(pOrigin,148.4,84.1,0.0),vDraw,z1,tPen\WObj:=wPaper;
    MoveL Offs(pOrigin,148.8,83.6,0.0),vDraw,z1,tPen\WObj:=wPaper;
    MoveL Offs(pOrigin,148.8,83.4,0.0),vDraw,z1,tPen\WObj:=wPaper;
    MoveL Offs(pOrigin,148.4,82.9,0.0),vDraw,fine,tPen\WObj:=wPaper;
    MoveL Offs(pOrigin,148.4,82.9,15.0),vApproach,z5,tPen\WObj:=wPaper;
    MoveL Offs(pOrigin,143.9,94.4,15.0),vTravel,z5,tPen\WObj:=wPaper;
    MoveL Offs(pOrigin,143.9,94.4,0.0),vApproach,fine,tPen\WObj:=wPaper;
    MoveL Offs(pOrigin,143.7,94.4,0.0),vDraw,z1,tPen\WObj:=wPaper;
    MoveL Offs(pOrigin,143.2,95.1,0.0),vDraw,z1,tPen\WObj:=wPaper;
    MoveL Offs(pOrigin,142.3,95.1,0.0),vDraw,z1,tPen\WObj:=wPaper;
    MoveL Offs(pOrigin,142.1,95.3,0.0),vDraw,z1,tPen\WObj:=wPaper;
    MoveL Offs(pOrigin,142.1,95.5,0.0),vDraw,z1,tPen\WObj:=wPaper;
    MoveL Offs(pOrigin,142.5,96.0,0.0),vDraw,z1,tPen\WObj:=wPaper;
    MoveL Offs(pOrigin,142.8,96.0,0.0),vDraw,z1,tPen\WObj:=wPaper;
    MoveL Offs(pOrigin,143.2,95.5,0.0),vDraw,z1,tPen\WObj:=wPaper;
    MoveL Offs(pOrigin,143.7,95.5,0.0),vDraw,z1,tPen\WObj:=wPaper;
    MoveL Offs(pOrigin,144.2,95.1,0.0),vDraw,z1,tPen\WObj:=wPaper;
    MoveL Offs(pOrigin,144.2,94.6,0.0),vDraw,z1,tPen\WObj:=wPaper;
    MoveL Offs(pOrigin,143.9,94.4,0.0),vDraw,fine,tPen\WObj:=wPaper;
    MoveL Offs(pOrigin,143.9,94.4,15.0),vApproach,z5,tPen\WObj:=wPaper;
    MoveL Offs(pOrigin,140.2,94.4,15.0),vTravel,z5,tPen\WObj:=wPaper;
    MoveL Offs(pOrigin,140.2,94.4,0.0),vApproach,fine,tPen\WObj:=wPaper;
    MoveL Offs(pOrigin,140.0,94.1,0.0),vDraw,z1,tPen\WObj:=wPaper;
    MoveL Offs(pOrigin,139.7,94.1,0.0),vDraw,z1,tPen\WObj:=wPaper;
    MoveL Offs(pOrigin,139.3,94.6,0.0),vDraw,z1,tPen\WObj:=wPaper;
    MoveL Offs(pOrigin,139.3,95.1,0.0),vDraw,z1,tPen\WObj:=wPaper;
    MoveL Offs(pOrigin,138.8,95.5,0.0),vDraw,z1,tPen\WObj:=wPaper;
    MoveL Offs(pOrigin,139.5,96.2,0.0),vDraw,z1,tPen\WObj:=wPaper;
    MoveL Offs(pOrigin,139.7,96.0,0.0),vDraw,z1,tPen\WObj:=wPaper;
    MoveL Offs(pOrigin,139.7,95.8,0.0),vDraw,z1,tPen\WObj:=wPaper;
    MoveL Offs(pOrigin,140.0,95.5,0.0),vDraw,z1,tPen\WObj:=wPaper;
    MoveL Offs(pOrigin,140.0,95.1,0.0),vDraw,z1,tPen\WObj:=wPaper;
    MoveL Offs(pOrigin,140.2,94.8,0.0),vDraw,z1,tPen\WObj:=wPaper;
    MoveL Offs(pOrigin,140.2,94.4,0.0),vDraw,fine,tPen\WObj:=wPaper;
    MoveL Offs(pOrigin,140.2,94.4,15.0),vApproach,z5,tPen\WObj:=wPaper;
    MoveL Offs(pOrigin,126.2,91.6,15.0),vTravel,z5,tPen\WObj:=wPaper;
    MoveL Offs(pOrigin,126.2,91.6,0.0),vApproach,fine,tPen\WObj:=wPaper;
    MoveL Offs(pOrigin,126.0,91.8,0.0),vDraw,z1,tPen\WObj:=wPaper;
    MoveL Offs(pOrigin,126.0,93.2,0.0),vDraw,z1,tPen\WObj:=wPaper;
    MoveL Offs(pOrigin,125.7,93.4,0.0),vDraw,z1,tPen\WObj:=wPaper;
    MoveL Offs(pOrigin,125.7,98.8,0.0),vDraw,z1,tPen\WObj:=wPaper;
    MoveL Offs(pOrigin,126.0,99.0,0.0),vDraw,z1,tPen\WObj:=wPaper;
    MoveL Offs(pOrigin,126.0,100.7,0.0),vDraw,z1,tPen\WObj:=wPaper;
    MoveL Offs(pOrigin,126.2,100.9,0.0),vDraw,z1,tPen\WObj:=wPaper;
    MoveL Offs(pOrigin,126.2,101.8,0.0),vDraw,z1,tPen\WObj:=wPaper;
    MoveL Offs(pOrigin,126.4,102.1,0.0),vDraw,z1,tPen\WObj:=wPaper;
    MoveL Offs(pOrigin,126.4,102.8,0.0),vDraw,z1,tPen\WObj:=wPaper;
    MoveL Offs(pOrigin,126.7,103.0,0.0),vDraw,z1,tPen\WObj:=wPaper;
    MoveL Offs(pOrigin,126.7,103.7,0.0),vDraw,z1,tPen\WObj:=wPaper;
    MoveL Offs(pOrigin,126.9,103.9,0.0),vDraw,z1,tPen\WObj:=wPaper;
    MoveL Offs(pOrigin,126.9,104.4,0.0),vDraw,z1,tPen\WObj:=wPaper;
    MoveL Offs(pOrigin,127.1,104.6,0.0),vDraw,z1,tPen\WObj:=wPaper;
    MoveL Offs(pOrigin,127.1,105.1,0.0),vDraw,z1,tPen\WObj:=wPaper;
    MoveL Offs(pOrigin,127.4,105.3,0.0),vDraw,z1,tPen\WObj:=wPaper;
    MoveL Offs(pOrigin,127.4,106.0,0.0),vDraw,z1,tPen\WObj:=wPaper;
    MoveL Offs(pOrigin,127.6,106.3,0.0),vDraw,z1,tPen\WObj:=wPaper;
    MoveL Offs(pOrigin,127.6,106.7,0.0),vDraw,z1,tPen\WObj:=wPaper;
    MoveL Offs(pOrigin,127.4,106.7,0.0),vDraw,z1,tPen\WObj:=wPaper;
    MoveL Offs(pOrigin,126.4,105.8,0.0),vDraw,z1,tPen\WObj:=wPaper;
    MoveL Offs(pOrigin,126.4,105.6,0.0),vDraw,z1,tPen\WObj:=wPaper;
    MoveL Offs(pOrigin,124.8,103.7,0.0),vDraw,z1,tPen\WObj:=wPaper;
    MoveL Offs(pOrigin,124.8,103.5,0.0),vDraw,z1,tPen\WObj:=wPaper;
    MoveL Offs(pOrigin,124.3,103.0,0.0),vDraw,z1,tPen\WObj:=wPaper;
    MoveL Offs(pOrigin,124.3,102.8,0.0),vDraw,z1,tPen\WObj:=wPaper;
    MoveL Offs(pOrigin,123.4,101.8,0.0),vDraw,z1,tPen\WObj:=wPaper;
    MoveL Offs(pOrigin,123.4,101.6,0.0),vDraw,z1,tPen\WObj:=wPaper;
    MoveL Offs(pOrigin,121.5,99.7,0.0),vDraw,z1,tPen\WObj:=wPaper;
    MoveL Offs(pOrigin,121.5,99.5,0.0),vDraw,z1,tPen\WObj:=wPaper;
    MoveL Offs(pOrigin,119.2,97.2,0.0),vDraw,z1,tPen\WObj:=wPaper;
    MoveL Offs(pOrigin,119.0,97.2,0.0),vDraw,z1,tPen\WObj:=wPaper;
    MoveL Offs(pOrigin,117.3,95.5,0.0),vDraw,z1,tPen\WObj:=wPaper;
    MoveL Offs(pOrigin,117.1,95.5,0.0),vDraw,z1,tPen\WObj:=wPaper;
    MoveL Offs(pOrigin,116.4,94.8,0.0),vDraw,z1,tPen\WObj:=wPaper;
    MoveL Offs(pOrigin,116.2,94.8,0.0),vDraw,z1,tPen\WObj:=wPaper;
    MoveL Offs(pOrigin,115.9,94.6,0.0),vDraw,z1,tPen\WObj:=wPaper;
    MoveL Offs(pOrigin,115.2,94.6,0.0),vDraw,z1,tPen\WObj:=wPaper;
    MoveL Offs(pOrigin,115.0,94.4,0.0),vDraw,z1,tPen\WObj:=wPaper;
    MoveL Offs(pOrigin,114.8,94.4,0.0),vDraw,z1,tPen\WObj:=wPaper;
    MoveL Offs(pOrigin,114.5,94.1,0.0),vDraw,z1,tPen\WObj:=wPaper;
    MoveL Offs(pOrigin,114.1,94.1,0.0),vDraw,z1,tPen\WObj:=wPaper;
    MoveL Offs(pOrigin,113.4,93.7,0.0),vDraw,z1,tPen\WObj:=wPaper;
    MoveL Offs(pOrigin,112.9,93.7,0.0),vDraw,z1,tPen\WObj:=wPaper;
    MoveL Offs(pOrigin,112.7,93.4,0.0),vDraw,z1,tPen\WObj:=wPaper;
    MoveL Offs(pOrigin,112.2,93.4,0.0),vDraw,z1,tPen\WObj:=wPaper;
    MoveL Offs(pOrigin,112.0,93.2,0.0),vDraw,z1,tPen\WObj:=wPaper;
    MoveL Offs(pOrigin,111.5,93.2,0.0),vDraw,z1,tPen\WObj:=wPaper;
  ENDPROC

  PROC Part17()
    MoveL Offs(pOrigin,111.3,93.0,0.0),vDraw,z1,tPen\WObj:=wPaper;
    MoveL Offs(pOrigin,110.1,92.7,0.0),vDraw,z1,tPen\WObj:=wPaper;
    MoveL Offs(pOrigin,109.4,92.3,0.0),vDraw,z1,tPen\WObj:=wPaper;
    MoveL Offs(pOrigin,108.7,92.3,0.0),vDraw,z1,tPen\WObj:=wPaper;
    MoveL Offs(pOrigin,108.0,91.8,0.0),vDraw,z1,tPen\WObj:=wPaper;
    MoveL Offs(pOrigin,107.5,91.8,0.0),vDraw,z1,tPen\WObj:=wPaper;
    MoveL Offs(pOrigin,107.3,91.6,0.0),vDraw,z1,tPen\WObj:=wPaper;
    MoveL Offs(pOrigin,106.8,91.6,0.0),vDraw,z1,tPen\WObj:=wPaper;
    MoveL Offs(pOrigin,106.6,91.3,0.0),vDraw,z1,tPen\WObj:=wPaper;
    MoveL Offs(pOrigin,105.4,91.1,0.0),vDraw,z1,tPen\WObj:=wPaper;
    MoveL Offs(pOrigin,104.7,90.6,0.0),vDraw,z1,tPen\WObj:=wPaper;
    MoveL Offs(pOrigin,104.3,90.6,0.0),vDraw,z1,tPen\WObj:=wPaper;
    MoveL Offs(pOrigin,104.0,90.4,0.0),vDraw,z1,tPen\WObj:=wPaper;
    MoveL Offs(pOrigin,103.8,90.4,0.0),vDraw,z1,tPen\WObj:=wPaper;
    MoveL Offs(pOrigin,103.6,90.2,0.0),vDraw,z1,tPen\WObj:=wPaper;
    MoveL Offs(pOrigin,103.1,90.2,0.0),vDraw,z1,tPen\WObj:=wPaper;
    MoveL Offs(pOrigin,102.4,89.7,0.0),vDraw,z1,tPen\WObj:=wPaper;
    MoveL Offs(pOrigin,101.2,89.5,0.0),vDraw,z1,tPen\WObj:=wPaper;
    MoveL Offs(pOrigin,100.5,89.0,0.0),vDraw,z1,tPen\WObj:=wPaper;
    MoveL Offs(pOrigin,99.4,88.8,0.0),vDraw,z1,tPen\WObj:=wPaper;
    MoveL Offs(pOrigin,99.1,88.5,0.0),vDraw,z1,tPen\WObj:=wPaper;
    MoveL Offs(pOrigin,98.9,88.5,0.0),vDraw,z1,tPen\WObj:=wPaper;
    MoveL Offs(pOrigin,98.7,88.3,0.0),vDraw,z1,tPen\WObj:=wPaper;
    MoveL Offs(pOrigin,98.2,88.3,0.0),vDraw,z1,tPen\WObj:=wPaper;
    MoveL Offs(pOrigin,97.5,87.8,0.0),vDraw,z1,tPen\WObj:=wPaper;
    MoveL Offs(pOrigin,97.0,87.8,0.0),vDraw,z1,tPen\WObj:=wPaper;
    MoveL Offs(pOrigin,96.8,87.6,0.0),vDraw,z1,tPen\WObj:=wPaper;
    MoveL Offs(pOrigin,95.6,87.4,0.0),vDraw,z1,tPen\WObj:=wPaper;
    MoveL Offs(pOrigin,94.9,86.9,0.0),vDraw,z1,tPen\WObj:=wPaper;
    MoveL Offs(pOrigin,94.5,86.9,0.0),vDraw,z1,tPen\WObj:=wPaper;
    MoveL Offs(pOrigin,94.2,86.7,0.0),vDraw,z1,tPen\WObj:=wPaper;
    MoveL Offs(pOrigin,93.5,86.7,0.0),vDraw,z1,tPen\WObj:=wPaper;
    MoveL Offs(pOrigin,92.8,86.2,0.0),vDraw,z1,tPen\WObj:=wPaper;
    MoveL Offs(pOrigin,92.4,86.2,0.0),vDraw,z1,tPen\WObj:=wPaper;
    MoveL Offs(pOrigin,92.1,86.0,0.0),vDraw,z1,tPen\WObj:=wPaper;
    MoveL Offs(pOrigin,91.7,86.0,0.0),vDraw,z1,tPen\WObj:=wPaper;
    MoveL Offs(pOrigin,91.4,85.7,0.0),vDraw,z1,tPen\WObj:=wPaper;
    MoveL Offs(pOrigin,91.0,85.7,0.0),vDraw,z1,tPen\WObj:=wPaper;
    MoveL Offs(pOrigin,90.7,85.5,0.0),vDraw,z1,tPen\WObj:=wPaper;
    MoveL Offs(pOrigin,90.3,85.5,0.0),vDraw,z1,tPen\WObj:=wPaper;
    MoveL Offs(pOrigin,90.0,85.3,0.0),vDraw,z1,tPen\WObj:=wPaper;
    MoveL Offs(pOrigin,89.6,85.3,0.0),vDraw,z1,tPen\WObj:=wPaper;
    MoveL Offs(pOrigin,89.3,85.0,0.0),vDraw,z1,tPen\WObj:=wPaper;
    MoveL Offs(pOrigin,88.9,85.0,0.0),vDraw,z1,tPen\WObj:=wPaper;
    MoveL Offs(pOrigin,88.6,84.8,0.0),vDraw,z1,tPen\WObj:=wPaper;
    MoveL Offs(pOrigin,88.2,84.8,0.0),vDraw,z1,tPen\WObj:=wPaper;
    MoveL Offs(pOrigin,87.9,84.6,0.0),vDraw,z1,tPen\WObj:=wPaper;
    MoveL Offs(pOrigin,87.5,84.6,0.0),vDraw,z1,tPen\WObj:=wPaper;
    MoveL Offs(pOrigin,87.2,84.3,0.0),vDraw,z1,tPen\WObj:=wPaper;
    MoveL Offs(pOrigin,86.8,84.3,0.0),vDraw,z1,tPen\WObj:=wPaper;
    MoveL Offs(pOrigin,86.5,84.1,0.0),vDraw,z1,tPen\WObj:=wPaper;
    MoveL Offs(pOrigin,86.1,84.1,0.0),vDraw,z1,tPen\WObj:=wPaper;
    MoveL Offs(pOrigin,85.8,83.9,0.0),vDraw,z1,tPen\WObj:=wPaper;
    MoveL Offs(pOrigin,85.4,83.9,0.0),vDraw,z1,tPen\WObj:=wPaper;
    MoveL Offs(pOrigin,85.1,83.6,0.0),vDraw,z1,tPen\WObj:=wPaper;
    MoveL Offs(pOrigin,84.0,83.4,0.0),vDraw,z1,tPen\WObj:=wPaper;
    MoveL Offs(pOrigin,83.3,82.9,0.0),vDraw,z1,tPen\WObj:=wPaper;
    MoveL Offs(pOrigin,82.8,82.9,0.0),vDraw,z1,tPen\WObj:=wPaper;
    MoveL Offs(pOrigin,82.6,82.7,0.0),vDraw,z1,tPen\WObj:=wPaper;
    MoveL Offs(pOrigin,81.4,82.5,0.0),vDraw,z1,tPen\WObj:=wPaper;
    MoveL Offs(pOrigin,80.7,82.0,0.0),vDraw,z1,tPen\WObj:=wPaper;
    MoveL Offs(pOrigin,80.2,82.0,0.0),vDraw,z1,tPen\WObj:=wPaper;
    MoveL Offs(pOrigin,79.5,81.5,0.0),vDraw,z1,tPen\WObj:=wPaper;
    MoveL Offs(pOrigin,79.1,81.5,0.0),vDraw,z1,tPen\WObj:=wPaper;
    MoveL Offs(pOrigin,78.4,81.1,0.0),vDraw,z1,tPen\WObj:=wPaper;
    MoveL Offs(pOrigin,77.9,81.1,0.0),vDraw,z1,tPen\WObj:=wPaper;
    MoveL Offs(pOrigin,76.3,80.1,0.0),vDraw,z1,tPen\WObj:=wPaper;
    MoveL Offs(pOrigin,75.8,80.1,0.0),vDraw,z1,tPen\WObj:=wPaper;
    MoveL Offs(pOrigin,74.6,79.4,0.0),vDraw,z1,tPen\WObj:=wPaper;
    MoveL Offs(pOrigin,74.2,79.4,0.0),vDraw,z1,tPen\WObj:=wPaper;
    MoveL Offs(pOrigin,73.9,79.2,0.0),vDraw,z1,tPen\WObj:=wPaper;
    MoveL Offs(pOrigin,73.2,79.0,0.0),vDraw,z1,tPen\WObj:=wPaper;
    MoveL Offs(pOrigin,72.8,78.5,0.0),vDraw,z1,tPen\WObj:=wPaper;
    MoveL Offs(pOrigin,72.5,78.5,0.0),vDraw,z1,tPen\WObj:=wPaper;
    MoveL Offs(pOrigin,72.3,78.7,0.0),vDraw,z1,tPen\WObj:=wPaper;
    MoveL Offs(pOrigin,71.1,78.5,0.0),vDraw,z1,tPen\WObj:=wPaper;
    MoveL Offs(pOrigin,69.5,76.9,0.0),vDraw,z1,tPen\WObj:=wPaper;
    MoveL Offs(pOrigin,69.5,76.6,0.0),vDraw,z1,tPen\WObj:=wPaper;
    MoveL Offs(pOrigin,69.0,75.9,0.0),vDraw,z1,tPen\WObj:=wPaper;
    MoveL Offs(pOrigin,68.8,74.8,0.0),vDraw,z1,tPen\WObj:=wPaper;
    MoveL Offs(pOrigin,68.6,74.5,0.0),vDraw,z1,tPen\WObj:=wPaper;
    MoveL Offs(pOrigin,68.6,73.6,0.0),vDraw,z1,tPen\WObj:=wPaper;
    MoveL Offs(pOrigin,68.3,73.4,0.0),vDraw,z1,tPen\WObj:=wPaper;
    MoveL Offs(pOrigin,68.3,72.7,0.0),vDraw,z1,tPen\WObj:=wPaper;
    MoveL Offs(pOrigin,68.1,72.4,0.0),vDraw,z1,tPen\WObj:=wPaper;
    MoveL Offs(pOrigin,68.1,5.2,0.0),vDraw,z1,tPen\WObj:=wPaper;
    MoveL Offs(pOrigin,141.8,5.2,0.0),vDraw,z1,tPen\WObj:=wPaper;
    MoveL Offs(pOrigin,141.8,5.9,0.0),vDraw,z1,tPen\WObj:=wPaper;
    MoveL Offs(pOrigin,141.6,6.2,0.0),vDraw,z1,tPen\WObj:=wPaper;
    MoveL Offs(pOrigin,141.6,7.1,0.0),vDraw,z1,tPen\WObj:=wPaper;
    MoveL Offs(pOrigin,141.4,7.3,0.0),vDraw,z1,tPen\WObj:=wPaper;
    MoveL Offs(pOrigin,141.4,8.0,0.0),vDraw,z1,tPen\WObj:=wPaper;
    MoveL Offs(pOrigin,141.1,8.3,0.0),vDraw,z1,tPen\WObj:=wPaper;
    MoveL Offs(pOrigin,141.1,9.0,0.0),vDraw,z1,tPen\WObj:=wPaper;
    MoveL Offs(pOrigin,140.9,9.2,0.0),vDraw,z1,tPen\WObj:=wPaper;
    MoveL Offs(pOrigin,140.9,10.1,0.0),vDraw,z1,tPen\WObj:=wPaper;
    MoveL Offs(pOrigin,140.7,10.4,0.0),vDraw,z1,tPen\WObj:=wPaper;
    MoveL Offs(pOrigin,140.7,11.1,0.0),vDraw,z1,tPen\WObj:=wPaper;
    MoveL Offs(pOrigin,140.4,11.3,0.0),vDraw,z1,tPen\WObj:=wPaper;
    MoveL Offs(pOrigin,140.4,12.0,0.0),vDraw,z1,tPen\WObj:=wPaper;
    MoveL Offs(pOrigin,140.2,12.2,0.0),vDraw,z1,tPen\WObj:=wPaper;
    MoveL Offs(pOrigin,140.2,13.2,0.0),vDraw,z1,tPen\WObj:=wPaper;
    MoveL Offs(pOrigin,140.0,13.4,0.0),vDraw,z1,tPen\WObj:=wPaper;
    MoveL Offs(pOrigin,140.0,14.1,0.0),vDraw,z1,tPen\WObj:=wPaper;
    MoveL Offs(pOrigin,139.7,14.3,0.0),vDraw,z1,tPen\WObj:=wPaper;
    MoveL Offs(pOrigin,139.7,15.3,0.0),vDraw,z1,tPen\WObj:=wPaper;
    MoveL Offs(pOrigin,139.5,15.5,0.0),vDraw,z1,tPen\WObj:=wPaper;
    MoveL Offs(pOrigin,139.5,16.2,0.0),vDraw,z1,tPen\WObj:=wPaper;
    MoveL Offs(pOrigin,139.3,16.4,0.0),vDraw,z1,tPen\WObj:=wPaper;
    MoveL Offs(pOrigin,139.3,17.4,0.0),vDraw,z1,tPen\WObj:=wPaper;
    MoveL Offs(pOrigin,139.0,17.6,0.0),vDraw,z1,tPen\WObj:=wPaper;
    MoveL Offs(pOrigin,139.0,18.3,0.0),vDraw,z1,tPen\WObj:=wPaper;
    MoveL Offs(pOrigin,138.8,18.5,0.0),vDraw,z1,tPen\WObj:=wPaper;
    MoveL Offs(pOrigin,138.8,19.5,0.0),vDraw,z1,tPen\WObj:=wPaper;
    MoveL Offs(pOrigin,138.6,19.7,0.0),vDraw,z1,tPen\WObj:=wPaper;
    MoveL Offs(pOrigin,138.6,20.4,0.0),vDraw,z1,tPen\WObj:=wPaper;
    MoveL Offs(pOrigin,138.3,20.6,0.0),vDraw,z1,tPen\WObj:=wPaper;
    MoveL Offs(pOrigin,138.3,21.3,0.0),vDraw,z1,tPen\WObj:=wPaper;
    MoveL Offs(pOrigin,138.1,21.6,0.0),vDraw,z1,tPen\WObj:=wPaper;
    MoveL Offs(pOrigin,138.1,22.5,0.0),vDraw,z1,tPen\WObj:=wPaper;
  ENDPROC

  PROC Part18()
    MoveL Offs(pOrigin,137.9,22.7,0.0),vDraw,z1,tPen\WObj:=wPaper;
    MoveL Offs(pOrigin,137.9,23.7,0.0),vDraw,z1,tPen\WObj:=wPaper;
    MoveL Offs(pOrigin,137.6,23.9,0.0),vDraw,z1,tPen\WObj:=wPaper;
    MoveL Offs(pOrigin,137.6,24.8,0.0),vDraw,z1,tPen\WObj:=wPaper;
    MoveL Offs(pOrigin,137.4,25.1,0.0),vDraw,z1,tPen\WObj:=wPaper;
    MoveL Offs(pOrigin,137.4,26.0,0.0),vDraw,z1,tPen\WObj:=wPaper;
    MoveL Offs(pOrigin,137.2,26.2,0.0),vDraw,z1,tPen\WObj:=wPaper;
    MoveL Offs(pOrigin,137.2,27.4,0.0),vDraw,z1,tPen\WObj:=wPaper;
    MoveL Offs(pOrigin,136.9,27.6,0.0),vDraw,z1,tPen\WObj:=wPaper;
    MoveL Offs(pOrigin,136.9,28.6,0.0),vDraw,z1,tPen\WObj:=wPaper;
    MoveL Offs(pOrigin,136.7,28.8,0.0),vDraw,z1,tPen\WObj:=wPaper;
    MoveL Offs(pOrigin,136.7,29.5,0.0),vDraw,z1,tPen\WObj:=wPaper;
    MoveL Offs(pOrigin,136.5,29.7,0.0),vDraw,z1,tPen\WObj:=wPaper;
    MoveL Offs(pOrigin,136.5,30.7,0.0),vDraw,z1,tPen\WObj:=wPaper;
    MoveL Offs(pOrigin,136.2,30.9,0.0),vDraw,z1,tPen\WObj:=wPaper;
    MoveL Offs(pOrigin,136.2,31.8,0.0),vDraw,z1,tPen\WObj:=wPaper;
    MoveL Offs(pOrigin,136.0,32.1,0.0),vDraw,z1,tPen\WObj:=wPaper;
    MoveL Offs(pOrigin,136.0,32.8,0.0),vDraw,z1,tPen\WObj:=wPaper;
    MoveL Offs(pOrigin,135.8,33.0,0.0),vDraw,z1,tPen\WObj:=wPaper;
    MoveL Offs(pOrigin,135.8,33.9,0.0),vDraw,z1,tPen\WObj:=wPaper;
    MoveL Offs(pOrigin,135.5,34.2,0.0),vDraw,z1,tPen\WObj:=wPaper;
    MoveL Offs(pOrigin,135.5,34.9,0.0),vDraw,z1,tPen\WObj:=wPaper;
    MoveL Offs(pOrigin,135.3,35.1,0.0),vDraw,z1,tPen\WObj:=wPaper;
    MoveL Offs(pOrigin,135.3,36.0,0.0),vDraw,z1,tPen\WObj:=wPaper;
    MoveL Offs(pOrigin,135.1,36.3,0.0),vDraw,z1,tPen\WObj:=wPaper;
    MoveL Offs(pOrigin,135.1,37.2,0.0),vDraw,z1,tPen\WObj:=wPaper;
    MoveL Offs(pOrigin,134.8,37.4,0.0),vDraw,z1,tPen\WObj:=wPaper;
    MoveL Offs(pOrigin,134.8,38.4,0.0),vDraw,z1,tPen\WObj:=wPaper;
    MoveL Offs(pOrigin,134.6,38.6,0.0),vDraw,z1,tPen\WObj:=wPaper;
    MoveL Offs(pOrigin,134.6,39.8,0.0),vDraw,z1,tPen\WObj:=wPaper;
    MoveL Offs(pOrigin,134.4,40.0,0.0),vDraw,z1,tPen\WObj:=wPaper;
    MoveL Offs(pOrigin,134.4,40.9,0.0),vDraw,z1,tPen\WObj:=wPaper;
    MoveL Offs(pOrigin,134.1,41.2,0.0),vDraw,z1,tPen\WObj:=wPaper;
    MoveL Offs(pOrigin,134.1,42.1,0.0),vDraw,z1,tPen\WObj:=wPaper;
    MoveL Offs(pOrigin,133.9,42.3,0.0),vDraw,z1,tPen\WObj:=wPaper;
    MoveL Offs(pOrigin,133.9,43.5,0.0),vDraw,z1,tPen\WObj:=wPaper;
    MoveL Offs(pOrigin,133.7,43.7,0.0),vDraw,z1,tPen\WObj:=wPaper;
    MoveL Offs(pOrigin,133.7,44.9,0.0),vDraw,z1,tPen\WObj:=wPaper;
    MoveL Offs(pOrigin,133.4,45.1,0.0),vDraw,z1,tPen\WObj:=wPaper;
    MoveL Offs(pOrigin,133.4,46.1,0.0),vDraw,z1,tPen\WObj:=wPaper;
    MoveL Offs(pOrigin,133.2,46.3,0.0),vDraw,z1,tPen\WObj:=wPaper;
    MoveL Offs(pOrigin,133.2,47.5,0.0),vDraw,z1,tPen\WObj:=wPaper;
    MoveL Offs(pOrigin,133.0,47.7,0.0),vDraw,z1,tPen\WObj:=wPaper;
    MoveL Offs(pOrigin,133.0,48.9,0.0),vDraw,z1,tPen\WObj:=wPaper;
    MoveL Offs(pOrigin,132.7,49.1,0.0),vDraw,z1,tPen\WObj:=wPaper;
    MoveL Offs(pOrigin,132.7,50.3,0.0),vDraw,z1,tPen\WObj:=wPaper;
    MoveL Offs(pOrigin,132.5,50.5,0.0),vDraw,z1,tPen\WObj:=wPaper;
    MoveL Offs(pOrigin,132.5,51.9,0.0),vDraw,z1,tPen\WObj:=wPaper;
    MoveL Offs(pOrigin,132.3,52.1,0.0),vDraw,z1,tPen\WObj:=wPaper;
    MoveL Offs(pOrigin,132.3,53.1,0.0),vDraw,z1,tPen\WObj:=wPaper;
    MoveL Offs(pOrigin,132.0,53.3,0.0),vDraw,z1,tPen\WObj:=wPaper;
    MoveL Offs(pOrigin,132.0,54.7,0.0),vDraw,z1,tPen\WObj:=wPaper;
    MoveL Offs(pOrigin,131.8,54.9,0.0),vDraw,z1,tPen\WObj:=wPaper;
    MoveL Offs(pOrigin,131.8,56.1,0.0),vDraw,z1,tPen\WObj:=wPaper;
    MoveL Offs(pOrigin,131.6,56.3,0.0),vDraw,z1,tPen\WObj:=wPaper;
    MoveL Offs(pOrigin,131.6,57.5,0.0),vDraw,z1,tPen\WObj:=wPaper;
    MoveL Offs(pOrigin,131.3,57.7,0.0),vDraw,z1,tPen\WObj:=wPaper;
    MoveL Offs(pOrigin,131.3,58.9,0.0),vDraw,z1,tPen\WObj:=wPaper;
    MoveL Offs(pOrigin,131.1,59.1,0.0),vDraw,z1,tPen\WObj:=wPaper;
    MoveL Offs(pOrigin,131.1,60.3,0.0),vDraw,z1,tPen\WObj:=wPaper;
    MoveL Offs(pOrigin,130.9,60.5,0.0),vDraw,z1,tPen\WObj:=wPaper;
    MoveL Offs(pOrigin,130.9,61.7,0.0),vDraw,z1,tPen\WObj:=wPaper;
    MoveL Offs(pOrigin,130.6,61.9,0.0),vDraw,z1,tPen\WObj:=wPaper;
    MoveL Offs(pOrigin,130.6,63.1,0.0),vDraw,z1,tPen\WObj:=wPaper;
    MoveL Offs(pOrigin,130.4,63.3,0.0),vDraw,z1,tPen\WObj:=wPaper;
    MoveL Offs(pOrigin,130.4,64.5,0.0),vDraw,z1,tPen\WObj:=wPaper;
    MoveL Offs(pOrigin,130.2,64.7,0.0),vDraw,z1,tPen\WObj:=wPaper;
    MoveL Offs(pOrigin,130.2,66.1,0.0),vDraw,z1,tPen\WObj:=wPaper;
    MoveL Offs(pOrigin,129.9,66.4,0.0),vDraw,z1,tPen\WObj:=wPaper;
    MoveL Offs(pOrigin,129.9,67.5,0.0),vDraw,z1,tPen\WObj:=wPaper;
    MoveL Offs(pOrigin,129.7,67.8,0.0),vDraw,z1,tPen\WObj:=wPaper;
    MoveL Offs(pOrigin,129.7,69.2,0.0),vDraw,z1,tPen\WObj:=wPaper;
    MoveL Offs(pOrigin,129.5,69.4,0.0),vDraw,z1,tPen\WObj:=wPaper;
    MoveL Offs(pOrigin,129.5,70.6,0.0),vDraw,z1,tPen\WObj:=wPaper;
    MoveL Offs(pOrigin,129.2,70.8,0.0),vDraw,z1,tPen\WObj:=wPaper;
    MoveL Offs(pOrigin,129.2,72.4,0.0),vDraw,z1,tPen\WObj:=wPaper;
    MoveL Offs(pOrigin,129.0,72.7,0.0),vDraw,z1,tPen\WObj:=wPaper;
    MoveL Offs(pOrigin,129.0,73.8,0.0),vDraw,z1,tPen\WObj:=wPaper;
    MoveL Offs(pOrigin,128.8,74.1,0.0),vDraw,z1,tPen\WObj:=wPaper;
    MoveL Offs(pOrigin,128.8,75.7,0.0),vDraw,z1,tPen\WObj:=wPaper;
    MoveL Offs(pOrigin,128.5,75.9,0.0),vDraw,z1,tPen\WObj:=wPaper;
    MoveL Offs(pOrigin,128.5,77.6,0.0),vDraw,z1,tPen\WObj:=wPaper;
    MoveL Offs(pOrigin,128.3,77.8,0.0),vDraw,z1,tPen\WObj:=wPaper;
    MoveL Offs(pOrigin,128.3,79.4,0.0),vDraw,z1,tPen\WObj:=wPaper;
    MoveL Offs(pOrigin,128.1,79.7,0.0),vDraw,z1,tPen\WObj:=wPaper;
    MoveL Offs(pOrigin,128.1,81.1,0.0),vDraw,z1,tPen\WObj:=wPaper;
    MoveL Offs(pOrigin,127.8,81.3,0.0),vDraw,z1,tPen\WObj:=wPaper;
    MoveL Offs(pOrigin,127.8,82.7,0.0),vDraw,z1,tPen\WObj:=wPaper;
    MoveL Offs(pOrigin,127.6,82.9,0.0),vDraw,z1,tPen\WObj:=wPaper;
    MoveL Offs(pOrigin,127.6,84.1,0.0),vDraw,z1,tPen\WObj:=wPaper;
    MoveL Offs(pOrigin,127.4,84.3,0.0),vDraw,z1,tPen\WObj:=wPaper;
    MoveL Offs(pOrigin,127.4,85.5,0.0),vDraw,z1,tPen\WObj:=wPaper;
    MoveL Offs(pOrigin,127.1,85.7,0.0),vDraw,z1,tPen\WObj:=wPaper;
    MoveL Offs(pOrigin,127.1,86.9,0.0),vDraw,z1,tPen\WObj:=wPaper;
    MoveL Offs(pOrigin,126.9,87.1,0.0),vDraw,z1,tPen\WObj:=wPaper;
    MoveL Offs(pOrigin,126.9,88.5,0.0),vDraw,z1,tPen\WObj:=wPaper;
    MoveL Offs(pOrigin,126.7,88.8,0.0),vDraw,z1,tPen\WObj:=wPaper;
    MoveL Offs(pOrigin,126.7,89.7,0.0),vDraw,z1,tPen\WObj:=wPaper;
    MoveL Offs(pOrigin,126.4,89.9,0.0),vDraw,z1,tPen\WObj:=wPaper;
    MoveL Offs(pOrigin,126.4,90.4,0.0),vDraw,z1,tPen\WObj:=wPaper;
    MoveL Offs(pOrigin,126.2,90.6,0.0),vDraw,z1,tPen\WObj:=wPaper;
    MoveL Offs(pOrigin,126.2,91.6,0.0),vDraw,fine,tPen\WObj:=wPaper;
    MoveL Offs(pOrigin,126.2,91.6,15.0),vApproach,z5,tPen\WObj:=wPaper;
    MoveL Offs(pOrigin,122.7,126.1,15.0),vTravel,z5,tPen\WObj:=wPaper;
    MoveL Offs(pOrigin,122.7,126.1,0.0),vApproach,fine,tPen\WObj:=wPaper;
    MoveL Offs(pOrigin,121.3,126.1,0.0),vDraw,z1,tPen\WObj:=wPaper;
    MoveL Offs(pOrigin,119.9,127.3,0.0),vDraw,z1,tPen\WObj:=wPaper;
    MoveL Offs(pOrigin,119.9,127.5,0.0),vDraw,z1,tPen\WObj:=wPaper;
    MoveL Offs(pOrigin,120.1,127.7,0.0),vDraw,z1,tPen\WObj:=wPaper;
    MoveL Offs(pOrigin,120.4,127.7,0.0),vDraw,z1,tPen\WObj:=wPaper;
    MoveL Offs(pOrigin,121.1,127.3,0.0),vDraw,z1,tPen\WObj:=wPaper;
    MoveL Offs(pOrigin,122.5,127.3,0.0),vDraw,z1,tPen\WObj:=wPaper;
    MoveL Offs(pOrigin,122.7,127.5,0.0),vDraw,z1,tPen\WObj:=wPaper;
    MoveL Offs(pOrigin,122.9,127.5,0.0),vDraw,z1,tPen\WObj:=wPaper;
    MoveL Offs(pOrigin,122.9,127.7,0.0),vDraw,z1,tPen\WObj:=wPaper;
    MoveL Offs(pOrigin,124.1,128.9,0.0),vDraw,z1,tPen\WObj:=wPaper;
    MoveL Offs(pOrigin,124.3,128.9,0.0),vDraw,z1,tPen\WObj:=wPaper;
    MoveL Offs(pOrigin,124.6,129.1,0.0),vDraw,z1,tPen\WObj:=wPaper;
    MoveL Offs(pOrigin,125.0,128.7,0.0),vDraw,z1,tPen\WObj:=wPaper;
    MoveL Offs(pOrigin,125.0,127.7,0.0),vDraw,z1,tPen\WObj:=wPaper;
  ENDPROC

  PROC Part19()
    MoveL Offs(pOrigin,123.6,126.3,0.0),vDraw,z1,tPen\WObj:=wPaper;
    MoveL Offs(pOrigin,122.9,126.3,0.0),vDraw,z1,tPen\WObj:=wPaper;
    MoveL Offs(pOrigin,122.7,126.1,0.0),vDraw,fine,tPen\WObj:=wPaper;
    MoveL Offs(pOrigin,122.7,126.1,15.0),vApproach,z5,tPen\WObj:=wPaper;
    MoveL Offs(pOrigin,122.7,130.1,15.0),vTravel,z5,tPen\WObj:=wPaper;
    MoveL Offs(pOrigin,122.7,130.1,0.0),vApproach,fine,tPen\WObj:=wPaper;
    MoveL Offs(pOrigin,122.0,130.8,0.0),vDraw,z1,tPen\WObj:=wPaper;
    MoveL Offs(pOrigin,122.0,132.6,0.0),vDraw,z1,tPen\WObj:=wPaper;
    MoveL Offs(pOrigin,122.2,132.9,0.0),vDraw,z1,tPen\WObj:=wPaper;
    MoveL Offs(pOrigin,123.4,132.6,0.0),vDraw,z1,tPen\WObj:=wPaper;
    MoveL Offs(pOrigin,123.9,132.2,0.0),vDraw,z1,tPen\WObj:=wPaper;
    MoveL Offs(pOrigin,123.9,131.9,0.0),vDraw,z1,tPen\WObj:=wPaper;
    MoveL Offs(pOrigin,123.4,131.5,0.0),vDraw,z1,tPen\WObj:=wPaper;
    MoveL Offs(pOrigin,123.4,131.2,0.0),vDraw,z1,tPen\WObj:=wPaper;
    MoveL Offs(pOrigin,122.7,130.1,0.0),vDraw,fine,tPen\WObj:=wPaper;
    MoveL Offs(pOrigin,122.7,130.1,15.0),vApproach,z5,tPen\WObj:=wPaper;
    MoveL Offs(pOrigin,121.1,133.6,15.0),vTravel,z5,tPen\WObj:=wPaper;
    MoveL Offs(pOrigin,121.1,133.6,0.0),vApproach,fine,tPen\WObj:=wPaper;
    MoveL Offs(pOrigin,120.6,133.6,0.0),vDraw,z1,tPen\WObj:=wPaper;
    MoveL Offs(pOrigin,119.9,134.3,0.0),vDraw,z1,tPen\WObj:=wPaper;
    MoveL Offs(pOrigin,120.1,134.5,0.0),vDraw,z1,tPen\WObj:=wPaper;
    MoveL Offs(pOrigin,120.4,134.5,0.0),vDraw,z1,tPen\WObj:=wPaper;
    MoveL Offs(pOrigin,121.3,133.8,0.0),vDraw,z1,tPen\WObj:=wPaper;
    MoveL Offs(pOrigin,121.1,133.6,0.0),vDraw,fine,tPen\WObj:=wPaper;
    MoveL Offs(pOrigin,121.1,133.6,15.0),vApproach,z5,tPen\WObj:=wPaper;
    MoveL Offs(pOrigin,119.2,135.7,15.0),vTravel,z5,tPen\WObj:=wPaper;
    MoveL Offs(pOrigin,119.2,135.7,0.0),vApproach,fine,tPen\WObj:=wPaper;
    MoveL Offs(pOrigin,118.7,136.1,0.0),vDraw,z1,tPen\WObj:=wPaper;
    MoveL Offs(pOrigin,118.7,137.8,0.0),vDraw,z1,tPen\WObj:=wPaper;
    MoveL Offs(pOrigin,119.0,138.0,0.0),vDraw,z1,tPen\WObj:=wPaper;
    MoveL Offs(pOrigin,119.2,137.8,0.0),vDraw,z1,tPen\WObj:=wPaper;
    MoveL Offs(pOrigin,119.2,136.8,0.0),vDraw,z1,tPen\WObj:=wPaper;
    MoveL Offs(pOrigin,119.4,136.6,0.0),vDraw,z1,tPen\WObj:=wPaper;
    MoveL Offs(pOrigin,119.4,135.9,0.0),vDraw,z1,tPen\WObj:=wPaper;
    MoveL Offs(pOrigin,119.2,135.7,0.0),vDraw,fine,tPen\WObj:=wPaper;
    MoveL Offs(pOrigin,119.2,135.7,15.0),vApproach,z5,tPen\WObj:=wPaper;
    MoveL Offs(pOrigin,119.0,138.0,15.0),vTravel,z5,tPen\WObj:=wPaper;
    MoveL Offs(pOrigin,119.0,138.0,0.0),vApproach,fine,tPen\WObj:=wPaper;
    MoveL Offs(pOrigin,118.7,138.2,0.0),vDraw,z1,tPen\WObj:=wPaper;
    MoveL Offs(pOrigin,118.7,139.9,0.0),vDraw,z1,tPen\WObj:=wPaper;
    MoveL Offs(pOrigin,119.0,140.1,0.0),vDraw,z1,tPen\WObj:=wPaper;
    MoveL Offs(pOrigin,119.0,140.8,0.0),vDraw,z1,tPen\WObj:=wPaper;
    MoveL Offs(pOrigin,119.2,141.0,0.0),vDraw,z1,tPen\WObj:=wPaper;
    MoveL Offs(pOrigin,119.2,141.5,0.0),vDraw,z1,tPen\WObj:=wPaper;
    MoveL Offs(pOrigin,119.7,142.2,0.0),vDraw,z1,tPen\WObj:=wPaper;
    MoveL Offs(pOrigin,119.7,142.9,0.0),vDraw,z1,tPen\WObj:=wPaper;
    MoveL Offs(pOrigin,119.9,143.1,0.0),vDraw,z1,tPen\WObj:=wPaper;
    MoveL Offs(pOrigin,119.9,145.5,0.0),vDraw,z1,tPen\WObj:=wPaper;
    MoveL Offs(pOrigin,120.1,145.7,0.0),vDraw,z1,tPen\WObj:=wPaper;
    MoveL Offs(pOrigin,120.1,146.2,0.0),vDraw,z1,tPen\WObj:=wPaper;
    MoveL Offs(pOrigin,120.6,146.6,0.0),vDraw,z1,tPen\WObj:=wPaper;
    MoveL Offs(pOrigin,121.3,146.6,0.0),vDraw,z1,tPen\WObj:=wPaper;
    MoveL Offs(pOrigin,121.5,146.4,0.0),vDraw,z1,tPen\WObj:=wPaper;
    MoveL Offs(pOrigin,121.3,146.6,0.0),vDraw,z1,tPen\WObj:=wPaper;
    MoveL Offs(pOrigin,121.3,147.1,0.0),vDraw,z1,tPen\WObj:=wPaper;
    MoveL Offs(pOrigin,121.1,147.3,0.0),vDraw,z1,tPen\WObj:=wPaper;
    MoveL Offs(pOrigin,121.3,147.6,0.0),vDraw,z1,tPen\WObj:=wPaper;
    MoveL Offs(pOrigin,121.8,147.6,0.0),vDraw,z1,tPen\WObj:=wPaper;
    MoveL Offs(pOrigin,122.0,147.3,0.0),vDraw,z1,tPen\WObj:=wPaper;
    MoveL Offs(pOrigin,122.7,147.1,0.0),vDraw,z1,tPen\WObj:=wPaper;
    MoveL Offs(pOrigin,123.4,146.4,0.0),vDraw,z1,tPen\WObj:=wPaper;
    MoveL Offs(pOrigin,123.4,146.2,0.0),vDraw,z1,tPen\WObj:=wPaper;
    MoveL Offs(pOrigin,123.6,145.9,0.0),vDraw,z1,tPen\WObj:=wPaper;
    MoveL Offs(pOrigin,123.6,145.5,0.0),vDraw,z1,tPen\WObj:=wPaper;
    MoveL Offs(pOrigin,123.9,145.2,0.0),vDraw,z1,tPen\WObj:=wPaper;
    MoveL Offs(pOrigin,123.9,144.5,0.0),vDraw,z1,tPen\WObj:=wPaper;
    MoveL Offs(pOrigin,123.6,144.3,0.0),vDraw,z1,tPen\WObj:=wPaper;
    MoveL Offs(pOrigin,123.4,144.3,0.0),vDraw,z1,tPen\WObj:=wPaper;
    MoveL Offs(pOrigin,122.2,145.7,0.0),vDraw,z1,tPen\WObj:=wPaper;
    MoveL Offs(pOrigin,122.2,144.5,0.0),vDraw,z1,tPen\WObj:=wPaper;
    MoveL Offs(pOrigin,122.0,144.3,0.0),vDraw,z1,tPen\WObj:=wPaper;
    MoveL Offs(pOrigin,122.0,143.6,0.0),vDraw,z1,tPen\WObj:=wPaper;
    MoveL Offs(pOrigin,122.2,143.4,0.0),vDraw,z1,tPen\WObj:=wPaper;
    MoveL Offs(pOrigin,123.2,143.4,0.0),vDraw,z1,tPen\WObj:=wPaper;
    MoveL Offs(pOrigin,123.4,143.1,0.0),vDraw,z1,tPen\WObj:=wPaper;
    MoveL Offs(pOrigin,123.4,142.9,0.0),vDraw,z1,tPen\WObj:=wPaper;
    MoveL Offs(pOrigin,122.9,142.4,0.0),vDraw,z1,tPen\WObj:=wPaper;
    MoveL Offs(pOrigin,121.3,142.4,0.0),vDraw,z1,tPen\WObj:=wPaper;
    MoveL Offs(pOrigin,119.4,140.6,0.0),vDraw,z1,tPen\WObj:=wPaper;
    MoveL Offs(pOrigin,119.4,139.6,0.0),vDraw,z1,tPen\WObj:=wPaper;
    MoveL Offs(pOrigin,119.2,139.4,0.0),vDraw,z1,tPen\WObj:=wPaper;
    MoveL Offs(pOrigin,119.2,138.2,0.0),vDraw,z1,tPen\WObj:=wPaper;
    MoveL Offs(pOrigin,119.0,138.0,0.0),vDraw,fine,tPen\WObj:=wPaper;
    MoveL Offs(pOrigin,119.0,138.0,15.0),vApproach,z5,tPen\WObj:=wPaper;
    MoveL Offs(pOrigin,122.9,137.5,15.0),vTravel,z5,tPen\WObj:=wPaper;
    MoveL Offs(pOrigin,122.9,137.5,0.0),vApproach,fine,tPen\WObj:=wPaper;
    MoveL Offs(pOrigin,123.2,137.8,0.0),vDraw,z1,tPen\WObj:=wPaper;
    MoveL Offs(pOrigin,123.2,138.5,0.0),vDraw,z1,tPen\WObj:=wPaper;
    MoveL Offs(pOrigin,123.4,138.7,0.0),vDraw,z1,tPen\WObj:=wPaper;
    MoveL Offs(pOrigin,123.4,138.9,0.0),vDraw,z1,tPen\WObj:=wPaper;
    MoveL Offs(pOrigin,123.6,139.2,0.0),vDraw,z1,tPen\WObj:=wPaper;
    MoveL Offs(pOrigin,123.9,139.2,0.0),vDraw,z1,tPen\WObj:=wPaper;
    MoveL Offs(pOrigin,124.1,138.9,0.0),vDraw,z1,tPen\WObj:=wPaper;
    MoveL Offs(pOrigin,124.1,137.8,0.0),vDraw,z1,tPen\WObj:=wPaper;
    MoveL Offs(pOrigin,123.4,136.8,0.0),vDraw,z1,tPen\WObj:=wPaper;
    MoveL Offs(pOrigin,122.9,137.5,0.0),vDraw,fine,tPen\WObj:=wPaper;
    MoveL Offs(pOrigin,122.9,137.5,15.0),vApproach,z5,tPen\WObj:=wPaper;
  ENDPROC

ENDMODULE
